TYPE ST_SectorsStatus :
STRUCT
	AllSectorsStatus : REFERENCE TO ARRAY[GC.MIN_SECTOR_CT..GC.MAX_SECTOR_CT] OF ST_SectorStatus;
END_STRUCT
END_TYPE

(* stored: Version 1.1.0.1
   DUT ST_SectorsStatus: Id {60740fba-0d1e-46ce-8220-14a2a060e3ef} *)
